(* IEC 61131-3 sources: traffic-lights/PLC_TrafficLights/Class/StringInternal (part 2) *)

          TmpFree(#pa, #thelp[0]);
        end_if;
      else
        // cat at end + termination
        tmp := chrcount * chrsize;
        if(TmpAlloc(#pa, tmp+2, #thelp[0], sizeof(thelp)) <> 0) then
          _memcpy(pa, psrc, tmp);
          pu  := pa + tmp;
          pu^ := 0; // do termination
          retcode := TxtCat(pa, chrsize); // concatenate
          TmpFree(#pa, #thelp[0]);
        end_if;
      end_if;
    end_if;
  end_if;

END_FUNCTION

FUNCTION VIRTUAL GLOBAL StringInternal::TxtToAscii
  VAR_OUTPUT
    retcode : bool;
  END_VAR
  VAR
  	pd : ^usint;
    len : udint;
  END_VAR

  retcode := true;

  pd := StrInt_GetData();
  if(pd <> nil) then
    if(StrInt_IsUnicode()) then
      len := TxtLen() + 1;
      if(len = 1) then
        KillUBOM();
      end_if;
      ToAsciiSequence(pd, pd$^uint+2, len, false);
      if(SingleRealloc = 0) then
        DataBuffer.SetSize(len);
      end_if;
      DataBuffer.UpdateToFile();
      m_udCRC := StrInt_CrcMakro(len);
    end_if;
  end_if;

END_FUNCTION

FUNCTION VIRTUAL GLOBAL StringInternal::TxtToUni
  VAR_OUTPUT
    retcode : bool;
  END_VAR
  VAR
    thelp : array[0..SI_TMP_HELPSIZE] of usint;
  	pd : ^usint;
    pu : ^uint;
    len : udint;
  END_VAR

  retcode := true;

  pd := StrInt_GetData();
  if(pd = nil) then
    retcode := TxtSet(2, "", 1);
  else
    if(StrInt_IsAscii()) then
      len := TxtLen() + 1;
      if(TmpAlloc(#pu, len*2+2, #thelp[0], sizeof(thelp)) <> 0) then
        pu^ := 16#0200;
        ToUniSequence(pu+2, pd, len, false);
        retcode := AddDataIntern(pu$^usint, len*2+2, 0);
        TmpFree(#pu, #thelp[0]);
      end_if;
    end_if;
  end_if;

END_FUNCTION

FUNCTION VIRTUAL GLOBAL StringInternal::TxtUpr
  VAR
    pa : ^usint;
    pu : ^uint;
    size : udint;
  END_VAR

	pa := StrInt_GetData();

  if(pa <> NIL) then
    if(StrInt_IsUnicode()) then
      pu   := pa$^uint + 2;
      size := 4; // 16#0200 + termination
      while(pu^) do
        if((pu^ >= 'a') & (pu^ <= 'z')) then
          pu^ -= 'a'-'A';
        end_if;
        pu   += 2;
        size += 2;
      end_while;
    else
			_strupr(pa);
      size := _strlen(pa) + 1;
    end_if;

    DataBuffer.UpdateToFile();
    m_udCrc := StrInt_CrcMakro(size);
	end_if;

END_FUNCTION

FUNCTION VIRTUAL GLOBAL StringInternal::TxtLwr
  VAR
    pu : ^uint;
    pa : ^usint;
    size : udint;
  END_VAR

	pa := StrInt_GetData();
  if(pa <> NIL) then
    if(StrInt_IsUnicode()) then
      pu   := pa$^uint + 2;
      size := 4; // 16#0200 + termination
      while(pu^) do
        if((pu^ <= 'Z') & (pu^ >= 'A')) then
          pu^ -= ('A'-'a');
        end_if;
        pu   += 2;
        size += 2;
      end_while;
    else
      size := 1; // termination
      while(pa^) do
        if((pa^ <= 'Z') & (pa^ >= 'A')) then
          pa^ -= ('A'-'a');
        end_if;
        pa   += 1;
        size += 1;
      end_while;
    end_if;

    DataBuffer.UpdateToFile();
    m_udCrc := StrInt_CrcMakro(size);
  end_if;

END_FUNCTION

FUNCTION VIRTUAL GLOBAL StringInternal::TxtGetCharSize
	VAR_OUTPUT
		retcode 	: USINT;
	END_VAR
  VAR
	  pu : ^uint;
  END_VAR

  retcode   := 1;
  pu$^usint := StrInt_GetData();
  if(pu <> NIL) then
    if(DataBuffer.GetSize() >= 2) then
      if(pu^ = 16#0200) then
        retcode := 2;
      end_if;
    end_if;
  end_if;

END_FUNCTION

FUNCTION VIRTUAL GLOBAL StringInternal::TxtGetCRC
	VAR_OUTPUT
		retcode 	: UDINT;
	END_VAR

  retcode := m_udCrc;

END_FUNCTION

FUNCTION VIRTUAL GLOBAL StringInternal::ObjCat
	VAR_INPUT
		pStr 	: ^StringInternal;
	END_VAR
	VAR_OUTPUT
		retcode 	: BOOL;
	END_VAR
  VAR
  	ps : ^usint;
    chrsize : udint;
  END_VAR

  retcode := true;

  if(pStr <> nil) then
    ps := pStr^.StrInt_GetData();
    if(ps <> nil) then
      chrsize := pStr^.TxtGetCharSize();
      retcode := TxtCat(ps, chrsize);
    end_if;
  end_if;

END_FUNCTION

FUNCTION VIRTUAL GLOBAL StringInternal::ObjCatAt
	VAR_INPUT
		chroffset 	: UDINT;
		pStr 	: ^StringInternal;
	END_VAR
	VAR_OUTPUT
		retcode 	: BOOL;
	END_VAR
  VAR
  	ps : ^usint;
    chrsize : udint;
  END_VAR

  retcode := true;

  if(pStr <> nil) then
    ps := pStr^.StrInt_GetData();
    if(ps <> nil) then
      chrsize := pStr^.TxtGetCharSize();
      retcode := TxtCatAt(chroffset, ps, chrsize);
    end_if;
  end_if;

END_FUNCTION

FUNCTION VIRTUAL GLOBAL StringInternal::ObjCpy
	VAR_INPUT
		pStr 	: ^StringInternal;
	END_VAR
	VAR_OUTPUT
		retcode 	: BOOL;
	END_VAR
  VAR
  	ps : ^usint;
    chrsize, dchrsiz : udint;
  END_VAR

  retcode := true;

  if(pStr <> nil) then
    ps      := pStr^.StrInt_GetData();
    chrsize := pStr^.TxtGetCharSize();
    dchrsiz := chrsize;
    if(StrInt_GetData() <> nil) then
      dchrsiz := TxtGetCharSize();
    end_if;

    retcode := TxtSet(dchrsiz, ps, chrsize);
  end_if;

END_FUNCTION

FUNCTION VIRTUAL GLOBAL StringInternal::ObjCpyFrom
	VAR_INPUT
		pStr 	: ^StringInternal;
		fromwhere 	: UDINT;
		nchar 	: UDINT;
	END_VAR
	VAR_OUTPUT
		retcode 	: BOOL;
	END_VAR
  VAR
    thelp : array[0..SI_TMP_HELPSIZE] of usint;
  	sln, tmp, chrsize, dchrsiz : udint;
    pa : ^usint;
  END_VAR

  sln := pStr^.TxtLen();
  if(nchar > sln) then
    nchar := sln; // truncate number of characters to get
  end_if;

  tmp := (sln + 1) * pStr^.TxtGetCharSize();
  if(TmpAlloc(#pa, tmp+2, #thelp[0], sizeof(thelp)) <> 0) then // +2 for possibly unicode-id
    chrsize := pStr^.TxtGetAt(pa+2, tmp, fromwhere, nchar);
    if(chrsize > 0) then
      dchrsiz := chrsize;
      if(StrInt_GetData() <> nil) then
        dchrsiz := TxtGetCharSize();
      end_if;

      if(dchrsiz = 2) & (chrsize = 2) then
        pa$^uint^ := 16#0200; // speedhack
        retcode   := TxtSet(2, pa, 2);
      else
        retcode := TxtSet(dchrsiz, pa+2, chrsize);
      end_if;
    end_if;
    TmpFree(#pa, #thelp[0]);
  end_if;

END_FUNCTION

FUNCTION VIRTUAL GLOBAL StringInternal::ObjClone
	VAR_INPUT
		pStr 	: ^StringInternal;
	END_VAR
	VAR_OUTPUT
		retcode 	: BOOL;
	END_VAR
  VAR
  	ps : ^usint;
    chrsize : udint;
  END_VAR

  retcode := true;

  if(pStr <> nil) then
    ps      := pStr^.StrInt_GetData();
    chrsize := pStr^.TxtGetCharSize();
    retcode := TxtSet(chrsize, ps, chrsize);
  end_if;

END_FUNCTION

FUNCTION VIRTUAL GLOBAL StringInternal::ObjCmp
	VAR_INPUT
		pStr 	: ^StringInternal;
	END_VAR
	VAR_OUTPUT
		udNotEqual 	: UDINT;
	END_VAR

  udNotEqual := TxtCmp(pStr^.StrInt_GetData(), pStr^.TxtGetCharSize());

END_FUNCTION

FUNCTION VIRTUAL GLOBAL StringInternal::ObjICmp
	VAR_INPUT
		pStr 	: ^StringInternal;
	END_VAR
	VAR_OUTPUT
		udNotEqual 	: UDINT;
	END_VAR

  udNotEqual := TxtICmp(pStr^.StrInt_GetData(), pStr^.TxtGetCharSize());

END_FUNCTION

FUNCTION VIRTUAL GLOBAL StringInternal::ObjIns
	VAR_INPUT
		index_at 	: UDINT;
		pStr 	: ^StringInternal;
		chrcount 	: UDINT;
	END_VAR
	VAR_OUTPUT
		retcode 	: BOOL;
	END_VAR
  VAR
  	ps : ^usint;
  END_VAR

  retcode := true;

  if(pStr <> nil) then
    ps := pStr^.StrInt_GetData();
    retcode := TxtIns(index_at, ps, pStr^.TxtGetCharSize(), chrcount);
  end_if;

END_FUNCTION

FUNCTION StringInternal::KillUBOM
  VAR
  	ubom : uint;
  END_VAR

  if(StrInt_IsUnicode()) then
    ubom := 0;
    DataBuffer.SetDataAt(#ubom$usint, 2, 0);
  end_if;

END_FUNCTION

FUNCTION GLOBAL StringInternal::TxtLenAsciiToUtf8
	VAR_INPUT
		src_ascii 	: ^char;
	END_VAR
	VAR_OUTPUT
		retcode 	: UDINT;
	END_VAR
  VAR
  	ps08 : ^USINT;
  END_VAR

  // compute length of given ASCII string in UTF8-Format
  // NOTE: same algorithm as in funktion TxtAsciiToUtf8

  retcode := 0;

  if(src_ascii <> nil) then
    ps08 := src_ascii$^USINT;
    while(ps08^) do
      if((ps08^) < 16#80) then
        retcode += 1;
      else
        retcode += 2;
      end_if;
      ps08 += 1;
    end_while;
  end_if;

END_FUNCTION

FUNCTION GLOBAL StringInternal::TxtLenUniToUtf8
	VAR_INPUT
		src_uni 	: ^UINT;
	END_VAR
	VAR_OUTPUT
		retcode 	: UDINT;
	END_VAR
  VAR
  	ps16 : ^UINT;
    chr : UINT;
  END_VAR

  // compute length of given UNICODE string in UTF8-Format
  // NOTE: same algorithm as in funktion TxtUniToUtf8

  retcode := 0;

  if(src_uni <> nil) then
    ps16 := src_uni$^UINT;
    while(ps16^) do
      chr  := ps16^;
      ps16 += 2;
      if(chr < 16#0080) then
        retcode += 1;
      elsif(chr < 16#0800) then
        retcode += 2;
      else
        retcode += 3;
      end_if;
    end_while;
  end_if;

END_FUNCTION

FUNCTION GLOBAL StringInternal::TxtLenUtf8ToAscii
	VAR_INPUT
		src_utf8 	: ^CHAR;
	END_VAR
	VAR_OUTPUT
		retcode 	: UDINT;
	END_VAR

  // compute textlength of given utf8 formatted string in ascii-format
  retcode := TxtLenUtf8ToUni(src_utf8);

END_FUNCTION

FUNCTION GLOBAL StringInternal::TxtLenUtf8ToUni
	VAR_INPUT
		src_utf8 	: ^CHAR;
	END_VAR
	VAR_OUTPUT
		retcode 	: UDINT;
	END_VAR
  VAR
    ps : ^USINT;
    follow : UDINT;
    chr : UINT;
  END_VAR

  // compute textlength of given utf8 formatted string in u16-format

  retcode := 0;

  if(src_utf8 <> nil) then
    ps := src_utf8$^USINT;

    while(ps^) do

      chr := ps^;
      ps += 1;

      if(chr AND 16#0080) then

        follow := 0;

        if((chr AND 16#00E0) = 16#00C0) then
          follow := 1; // 1 folgebyte
        elsif((chr AND 16#00F0) = 16#00E0) then
          follow := 2; // 2 folgebytes
        elsif((chr AND 16#00F8) = 16#00F0) then
          follow := 3; // 3 folgebytes
        end_if;

        while(follow <> 0) do
          follow -= 1;

          if((ps^ AND 16#C0) = 16#80) then
            ps += 1;
            if(follow = 0) then
              retcode += 1;
            end_if;
          end_if;
        end_while;

      else
        retcode += 1;
      end_if;
    end_while;
  end_if;

END_FUNCTION

FUNCTION GLOBAL StringInternal::TxtAsciiToUtf8
	VAR_INPUT
		dst_utf8 	: ^CHAR;
		src_ascii 	: ^CHAR;
	END_VAR
	VAR_OUTPUT
		retcode 	: UDINT;
	END_VAR
  VAR
  	ps : ^USINT;
    pd : ^USINT;
    chr : USINT;
  END_VAR

  // NOTE: same algorithm as in funktion TxtLenUTF8

  retcode := 0;

  if(dst_utf8 <> nil) then
    pd := dst_utf8$^USINT;

    if(src_ascii <> nil) then
      ps := src_ascii$^USINT;

      while(ps^) do

        chr := ps^;
        ps  += 1;
        if(chr < 16#0080) then
          pd^  := chr$USINT;
          pd += 1;
          retcode += 1;
        else
          pd^    := to_usint(16#00C0 OR (chr SHR 6));
          pd += 1;
          pd^    := to_usint(16#0080 OR (chr AND 16#003F));
          pd += 1;
          retcode += 2;
        end_if;
      end_while;
    end_if;

    pd^ := 0;
  end_if;

END_FUNCTION

FUNCTION GLOBAL StringInternal::TxtUniToUtf8
	VAR_INPUT
		dst_utf8 	: ^CHAR;
		src_uni 	: ^UINT;
	END_VAR
	VAR_OUTPUT
		retcode 	: UDINT;
	END_VAR
  VAR
    pd : ^USINT;
    chr : UINT;
  END_VAR

  // convert unicode-0-string to utf8-0-string, function will return number of used bytes in destination, excluding final zero
  // NOTE: same algorithm as in funktion TxtLenUTF8

  retcode := 0;

  if(dst_utf8 <> nil) then
    pd := dst_utf8$^USINT;

    if(src_uni <> nil) then
      while(src_uni^) do

        chr := src_uni^;
        src_uni += 2;

        if(chr < 16#0080) then
          pd^ := chr$USINT;
          pd += 1;
          retcode += 1;
        elsif(chr < 16#0800) then
          pd^ := to_usint(16#00C0 OR (chr SHR 6));
          pd += 1;
          pd^ := to_usint(16#0080 OR (chr AND 16#003F));
          pd += 1;
          retcode += 2;
        else
          pd^ := to_usint(16#00E0 OR (chr SHR 12));
          pd += 1;
          pd^ := to_usint(16#0080 OR ((chr SHR 6) AND 16#003F));
          pd += 1;
          pd^ := to_usint(16#0080 OR (chr AND 16#003F));
          pd += 1;
          retcode += 3;
        end_if;

      end_while;
    end_if;

    pd^ := 0;
  end_if;

END_FUNCTION

FUNCTION GLOBAL StringInternal::TxtUtf8ToAscii
	VAR_INPUT
		dst_ascii 	: ^CHAR;
		src_utf8 	: ^CHAR;
	END_VAR
	VAR_OUTPUT
		retcode 	: UDINT;
	END_VAR
  VAR
  	ps : ^USINT;
    pd : ^USINT;
    follow : UDINT;
    chr : UINT;
  END_VAR

  retcode := 0;

  if(dst_ascii <> nil) then
    pd := dst_ascii$^USINT;

    if(src_utf8 <> nil) then
      ps := src_utf8$^USINT;

      while(ps^) do

        chr := ps^;
        ps  += 1;
        if(chr AND 0x0080) then
          follow := 0;
          if ((chr AND 16#00E0) = 16#00C0) then
            follow := 1; // 1 folgebyte
            chr    := chr AND 16#001F;
          elsif((chr AND 16#00F0) = 16#00E0) then
            follow := 2; // 2 folgebytes
            chr    := chr AND 16#000F;
          elsif((chr AND 16#00F8) = 16#00F0) then
            follow := 3; // 3 folgebytes
            chr    := chr AND 16#0007;
          end_if;

          while(follow <> 0) do
            follow -= 1;
            if((ps^ AND 16#C0) = 16#80) then
              chr := ((chr SHL 6) OR ((ps^) AND 16#3F));
              ps += 1;
              if(follow = 0) then
                if(chr > 255) then
                  chr := 63; //'?'
                end_if;
                pd^ := chr$usint;
                pd  += 1;
                retcode += 1;
              end_if;
            end_if;
          end_while;
        else
          pd^ := chr$usint;
          pd  += 1;
          retcode += 1;
        end_if;
      end_while;
    end_if;

    pd^ := 0;
  end_if;

END_FUNCTION

FUNCTION GLOBAL StringInternal::TxtUtf8ToUni
	VAR_INPUT
		dst_uni 	: ^UINT;
		src_utf8 	: ^CHAR;
	END_VAR
	VAR_OUTPUT
		retcode 	: UDINT;
	END_VAR
  VAR
    ps : ^USINT;
    follow : UDINT;
    chr : UINT;
  END_VAR

  // convert utf8-0-string to unicode-0-string, function will return number of characters in destination

  retcode := 0;
  if(dst_uni <> nil) then

    if(src_utf8 <> nil) then
      ps := src_utf8$^USINT;

      while(ps^) do

        chr := ps^;
        ps += 1;

        if(chr AND 16#0080) then

          follow := 0;

          if((chr AND 16#00E0) = 16#00C0) then
            follow := 1; // 1 folgebyte
            chr    := chr AND 16#001F;
          elsif((chr AND 16#00F0) = 16#00E0) then
            follow := 2; // 2 folgebytes
            chr    := chr AND 0x000F;
          elsif((chr AND 16#00F8) = 16#00F0) then
            follow := 3; // 3 folgebytes
            chr    := chr AND 16#0007;
          end_if;

          while(follow <> 0) do
            follow -= 1;

            if((ps^ AND 16#C0) = 16#80) then
              chr := ((chr SHL 6) OR (ps^ AND 16#3F));
              ps += 1;
              if (follow = 0) then
                dst_uni^ := chr;
                dst_uni += 2;
                retcode += 1;
              end_if;
            end_if;
          end_while;

        else
          dst_uni^ := chr;
          dst_uni += 2;
          retcode += 1;
        end_if;

      end_while;
    end_if;

    dst_uni^ := 0;
  end_if;

END_FUNCTION

FUNCTION VIRTUAL GLOBAL StringInternal::TxtSetUtf8
	VAR_INPUT
		src_utf8 	: ^CHAR;
	END_VAR
	VAR_OUTPUT
		retcode 	: BOOL;
	END_VAR
  VAR
  	tmplen : udint;
    pu : ^uint;
    thelp : array[0..SI_TMP_HELPSIZE] of uint;
  END_VAR

  retcode := false;
  tmplen  := (TxtLenUtf8ToUni(src_utf8) + 2) * 2; // final zero + unicode mark

  if(TmpAlloc(#pu, tmplen, #thelp[0], sizeof(thelp)) <> 0) then
    pu^ := 16#0200;
    TxtUtf8ToUni(pu+2, src_utf8);
    retcode := AddDataIntern(pu$^usint, tmplen, 0);
    TmpFree(#pu, #thelp[0]);
  end_if;

END_FUNCTION

FUNCTION VIRTUAL GLOBAL StringInternal::TxtGetUtf8
	VAR_INPUT
		dst_utf8 	: ^CHAR;
	END_VAR
	VAR_OUTPUT
		retcode 	: UDINT;
	END_VAR
  VAR
  	pa : ^usint;
  END_VAR

  retcode := 0;

  if(dst_utf8 <> nil) then
    pa        := StrInt_GetData();
    dst_utf8^ := 0;

    if(pa <> nil) then
      if(StrInt_IsUnicode()) then
        retcode := TxtUniToUtf8(dst_utf8, 2 + pa$^uint);
      else
        retcode := TxtAsciiToUtf8(dst_utf8, pa);
      end_if;
    end_if;
  end_if;

END_FUNCTION

FUNCTION VIRTUAL GLOBAL StringInternal::TxtLenUtf8
	VAR_OUTPUT
		retcode 	: UDINT;
	END_VAR
  VAR
  	ph : ^usint;
  END_VAR

  retcode := 0;
  ph      := StrInt_GetData();
  if(ph <> nil) then
    if(StrInt_IsUnicode()) then
      retcode := TxtLenUniToUtf8(2 + ph$^uint);
    else
      retcode := TxtLenAsciiToUtf8(ph);
    end_if;
  end_if;

END_FUNCTION

//FUNCTION GLOBAL StringInternal::TxtLen16
//	VAR_INPUT
//    src16 : ^uint;
//	END_VAR
//	VAR_OUTPUT
//		retcode 	: UDINT;
//	END_VAR
//
//  retcode := 0;
//  if(src16 <> nil) then
//    retcode := StrInt_StrLen16(src16);
//  end_if;
//
//END_FUNCTION
//
//FUNCTION GLOBAL StringInternal::TxtLen08
//	VAR_INPUT
//    src08 : ^char;
//	END_VAR
//	VAR_OUTPUT
//		retcode 	: UDINT;
//	END_VAR
//
//  retcode := 0;
//  if(src08 <> nil) then
//    retcode := _strlen(src08);
//  end_if;
//
//END_FUNCTION
//
//FUNCTION GLOBAL StringInternal::TxtNCpy16
//	VAR_INPUT
//    pd : ^uint;
//    ps : ^uint;
//    maxlen : udint;
//	END_VAR
//	VAR_OUTPUT
//		retcode 	: ^uint;
//	END_VAR
//
//  retcode := pd;
//  if((pd <> nil) & (ps <> nil)) then
//    StrInt_StrNCpy16(pd, ps, maxlen);
//  end_if;
//
//END_FUNCTION
//
//FUNCTION GLOBAL StringInternal::TxtNCpy08
//	VAR_INPUT
//    pd : ^char;
//    ps : ^char;
//    maxlen : udint;
//	END_VAR
//	VAR_OUTPUT
//		retcode 	: ^char;
//	END_VAR
//
//  retcode := pd;
//  if((pd <> nil) & (ps <> nil)) then
//    StrInt_StrNCpy08(pd&^usint; ps$^usint; maxlen);
//  end_if;
//
//END_FUNCTION
